{attribute addProperty BoxType "EL4134-0000-1016"}
{attribute addProperty Id "AO_Output_ChannelAT %Q*ARRAY[0..3] OF AO_Output_Channel_F57FA4F96480WcStateAT %I*WcState_64F6A8C6810InfoDataAT %I*InfoData_BC63D37F80100"}
{attribute addProperty CRC "1637824629"}
{attribute addProperty SizeInBites "152"}
{attribute addProperty SizeInBytes "19"}
TYPE EL4134_57EE2D9D :
STRUCT
	{attribute addProperty Name "AO_Output_Channel"}
	AO_Output_Channel : ARRAY[0..3] OF AO_Output_Channel_F57FA4F9;
	{attribute addProperty Name "WcState"}
	WcState : WcState_64F6A8C6;
	{attribute addProperty Name "InfoData"}
	InfoData : InfoData_BC63D37F;
END_STRUCT
END_TYPE

(* stored: Version 1.2.0.0, ProductVersion 3.1.4024.9
   DUT EL4134_57EE2D9D: Id {7cc5a2fd-c8f2-4eee-877a-e2f90694af9b} *)
